// TwinCAT 3 PLC project TestProject
// ProgramVersion: 3.1.4023.0
// libraries:
//   Tc2_Standard, * (Beckhoff Automation GmbH)
//   Tc2_System, * (Beckhoff Automation GmbH)
//   Tc3_Module, * (Beckhoff Automation GmbH)
//   BeckhoffJsonReadWriter,1.0,fbarresi
// project tree:
//   DUTs/ json_st.TcDUT, ParserMethod.TcDUT
//   / PlcTask.TcTTO
//   POUs/ MAIN.TcPOU

CONFIGURATION TestProject
    RESOURCE PLC ON TwinCAT3
        TASK PlcTask(INTERVAL := T#10ms, PRIORITY := 20);
        PROGRAM MAIN WITH PlcTask : MAIN;
    END_RESOURCE
END_CONFIGURATION

// ---- DUTs/json_st.TcDUT
TYPE json_st :
STRUCT
	{attribute 'json' := 'name'}
	name : STRING;
	{attribute 'json' := 'age'}
	age : INT;
	{attribute 'json' := 'car'}
	car : STRING;
END_STRUCT
END_TYPE

// ---- DUTs/ParserMethod.TcDUT
{attribute 'qualified_only'}
{attribute 'strict'}
{attribute 'to_string'}
TYPE ParserMethod :
(
    ReadFile,
    WriteFile
);
END_TYPE

// ---- POUs/MAIN.TcPOU
PROGRAM MAIN
VAR
	parser : JsonParser;
    json : json_st := (name:='test', age:=23, car := 'supercar');
	fileMethod : ParserMethod := ParserMethod.WriteFile;
	runExecute : BOOL;
	hasError : BOOL;
	errorId : UDINT;
	filename : STRING := 'test.json';
END_VAR

parser(
	Execute:=runExecute, 
	File:= CONCAT('C:/testing/', filename), 
	ParseMethod:= TO_STRING(fileMethod),
	Content:= 'MAIN.json',
	Port := 851,
	HasError=> hasError, 
	ErrorId=> errorId);
	
IF runExecute THEN
	runExecute := FALSE;
END_IF

END_PROGRAM
